SUBAPPLICATION mapping_AUX (* Subapplication Type *)
  (* Standard: 61499-2 *)
  (* Version 1.0, 2023-02-07, franz *)
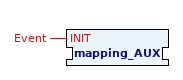
  EVENT_INPUT
    INIT;
  END_EVENT
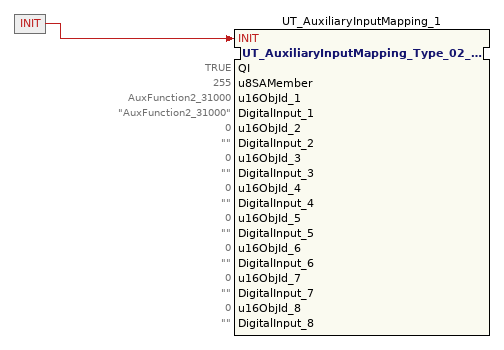
  FBS
    UT_AuxiliaryInputMapping_1 : UT_AuxiliaryInputMapping_Type_02_Bool_NonLatched(QI := TRUE, u8SAMember := 255, u16ObjId_1 := AuxFunction2_31000, DigitalInput_1 := "AuxFunction2_31000", u16ObjId_2 := 0, DigitalInput_2 := "", u16ObjId_3 := 0, DigitalInput_3 := "", u16ObjId_4 := 0, DigitalInput_4 := "", u16ObjId_5 := 0, DigitalInput_5 := "", u16ObjId_6 := 0, DigitalInput_6 := "", u16ObjId_7 := 0, DigitalInput_7 := "", u16ObjId_8 := 0, DigitalInput_8 := "");
  END_FBS
  EVENT_CONNECTIONS
    INIT TO UT_AuxiliaryInputMapping_1.INIT;
  END_CONNECTIONS
END_SUBAPPLICATION
